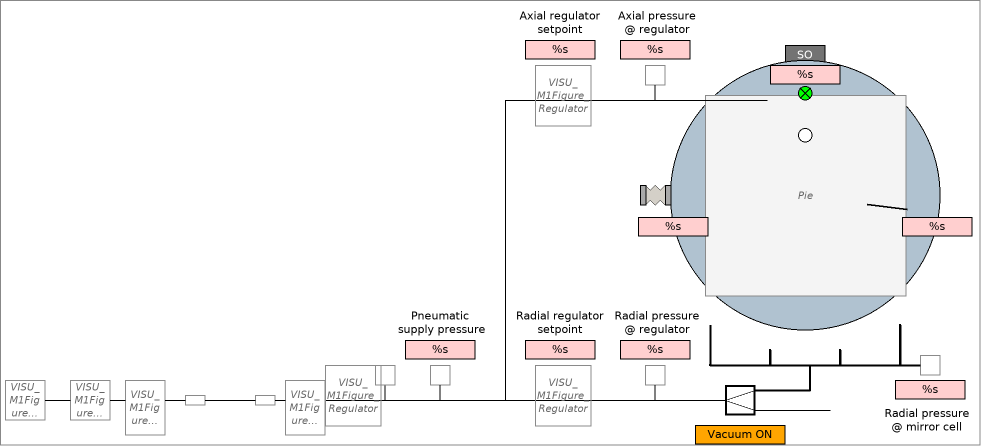
VISUALIZATION VISU_M1Figure  // 981x446
VAR_IN_OUT
	ref : M1;
    widget : M1Widget;
END_VAR
    Rectangle (785,45 40x33), "NW"
        p2858320360: widget.figure.axialNorthWestAngle
    Rectangle (785,45 40x30), "NE"
        p2858320360: widget.figure.axialNorthEastAngle
    Rectangle (785,45 40x33), "SO"
        p2858320360: widget.figure.axialSouthAngle
    Ellipse (670,60 270x270)
    Ellipse (770,160 70x70)
    Frame (920,355 20x20)
        shows VISU_M1Figure_Gauge()
    Rectangle (895,380 70x19), "%s", text variable: widget.figure.radialMirrorPressureString, colour variable: widget.radialSupport.mirrorPressure.actualStatusWidget.color.bg
        p55702900: widget.radialSupport.mirrorPressure.actualStatusWidget.color.fg
    Label (875,400 104x40), "Radial pressure @ mirror cell"
    Rectangle (725,385 30x30)
    Polyline (710,325) (710,365) (770,365) (770,350) (770,365) (840,365) (840,350) (840,365) (900,365) (900,325) (900,365) (920,365)
    Polyline (755,390) (810,390) (810,365)
    Rectangle (695,425 90x19), "Vacuum OFF", invisible if: ref.parts.radialSupport.parts.vacuumRelay.digitalOutput
    Line (755,410) (810,410)
    Line (810,410) (830,410)
    Line (725,400) (755,390), invisible if: ref.parts.radialSupport.parts.vacuumRelay.digitalOutput
    Line (725,400) (755,410), invisible if: NOT ref.parts.radialSupport.parts.vacuumRelay.digitalOutput
    Line (325,400) (725,400)
    Rectangle (665,185 6x20)
        p2858320360: widget.figure.radPad0Angle
    Polygon (650,200) (645,205) (645,185) (650,190) (655,185) (660,190) (665,185) (665,205) (660,200) (655,205)
        p2858320360: widget.figure.radPad0Angle
    Rectangle (640,185 6x20)
        p2858320360: widget.figure.radPad0Angle
    Rectangle (665,185 6x20)
        p2858320360: widget.figure.radPad1Angle
    Polygon (650,200) (645,205) (645,185) (650,190) (655,185) (660,190) (665,185) (665,205) (660,200) (655,205)
        p2858320360: widget.figure.radPad1Angle
    Rectangle (640,185 6x20)
        p2858320360: widget.figure.radPad1Angle
    Rectangle (665,185 6x20)
        p2858320360: widget.figure.radPad2Angle
    Polygon (650,200) (645,205) (645,185) (650,190) (655,185) (660,190) (665,185) (665,205) (660,200) (655,205)
        p2858320360: widget.figure.radPad2Angle
    Rectangle (640,185 6x20)
        p2858320360: widget.figure.radPad2Angle
    Rectangle (665,185 6x20)
        p2858320360: widget.figure.radPad3Angle
    Polygon (650,200) (645,205) (645,185) (650,190) (655,185) (660,190) (665,185) (665,205) (660,200) (655,205)
        p2858320360: widget.figure.radPad3Angle
    Rectangle (640,185 6x20)
        p2858320360: widget.figure.radPad3Angle
    Ellipse (744,135 123x123)
    Pie (705,95 201x201)
    Polyline (867,204) (907,209)
        p2858320360: widget.figure.axialSouthAngle
    Pie (705,95 201x201)
    Polyline (867,204) (907,209)
        p2858320360: widget.figure.axialNorthEastAngle
    Pie (705,95 201x201)
    Polyline (867,204) (907,209)
        p2858320360: widget.figure.axialNorthWestAngle
    Ellipse (798,128 14x14)
        p2858320360: widget.figure.axPadInner0Angle
    Ellipse (798,128 14x14)
        p2858320360: widget.figure.axPadInner1Angle
    Ellipse (798,128 14x14)
        p2858320360: widget.figure.axPadInner2Angle
    Ellipse (798,128 14x14)
        p2858320360: widget.figure.axPadInner3Angle
    Ellipse (798,128 14x14)
        p2858320360: widget.figure.axPadInner4Angle
    Ellipse (798,128 14x14)
        p2858320360: widget.figure.axPadInner5Angle
    Rectangle (770,65 70x19), "%s", text variable: widget.figure.axialForceStringSO, colour variable: widget.axialSupport.mirrorSouthForce.actualStatusWidget.color.bg
        p55702900: widget.axialSupport.mirrorSouthForce.actualStatusWidget.color.fg
    Rectangle (638,217 70x19), "%s", text variable: widget.figure.axialForceStringNW, colour variable: widget.axialSupport.mirrorNorthWestForce.actualStatusWidget.color.bg
        p55702900: widget.axialSupport.mirrorNorthWestForce.actualStatusWidget.color.fg
    Rectangle (902,217 70x19), "%s", text variable: widget.figure.axialForceStringNE, colour variable: widget.axialSupport.mirrorNorthEastForce.actualStatusWidget.color.bg
    Ellipse (798,86 14x14)
        p2858320360: widget.figure.axPad0Angle
    Ellipse (798,86 14x14)
        p2858320360: widget.figure.axPad1Angle
    Ellipse (798,86 14x14)
        p2858320360: widget.figure.axPad2Angle
    Ellipse (798,86 14x14)
        p2858320360: widget.figure.axPad3Angle
    Ellipse (798,86 14x14)
        p2858320360: widget.figure.axPad4Angle
    Ellipse (798,86 14x14)
        p2858320360: widget.figure.axPad5Angle
    Ellipse (798,86 14x14)
        p2858320360: widget.figure.axPad6Angle
    Ellipse (798,86 14x14)
        p2858320360: widget.figure.axPad7Angle
    Ellipse (798,86 14x14)
        p2858320360: widget.figure.axPad8Angle
    Ellipse (798,86 14x14), colour variable: widget.axialSupport.mirrorSouthForce.actualStatusWidget.color.bg
        p2858320360: widget.figure.axialSouthAngle
        p55702900: widget.axialSupport.mirrorSouthForce.actualStatusWidget.color.bg
    Polyline (810,98) (800,88)
        p2858320360: widget.figure.axialSouthAngle
    Polyline (810,88) (800,98)
        p2858320360: widget.figure.axialSouthAngle
    Ellipse (798,86 14x14), colour variable: widget.axialSupport.mirrorNorthEastForce.actualStatusWidget.color.bg
        p2858320360: widget.figure.axialNorthEastAngle
    Polyline (810,98) (800,88)
        p2858320360: widget.figure.axialNorthEastAngle
    Polyline (810,88) (800,98)
        p2858320360: widget.figure.axialNorthEastAngle
    Ellipse (798,86 14x14), colour variable: widget.axialSupport.mirrorNorthWestForce.actualStatusWidget.color.bg
        p2858320360: widget.figure.axialNorthWestAngle
    Polyline (810,98) (800,88)
        p2858320360: widget.figure.axialNorthWestAngle
    Polyline (810,88) (800,98)
        p2858320360: widget.figure.axialNorthWestAngle
    Line (505,100) (767,100)
    Frame (645,65 20x20)
        shows VISU_M1Figure_Gauge()
    Line (655,100) (655,85)
    Rectangle (620,40 70x19), "%s", text variable: widget.figure.axialRegulatorPressureString, colour variable: widget.axialSupport.regulatorPressure.actualStatusWidget.color.bg
        p55702900: widget.axialSupport.regulatorPressure.actualStatusWidget.color.fg
    Label (605,5 104x35), "Axial pressure @ regulator"
    Frame (535,65 56x61)
        shows VISU_M1Figure_Regulator()
    Label (515,5 90x35), "Axial regulator setpoint"
    Rectangle (525,40 70x19), "%s", text variable: widget.figure.axialRegulatorSetpointString, colour variable: widget.axialSupport.actualStatus.color.bg
        p55702900: widget.axialSupport.actualStatus.color.fg
    Frame (645,365 20x20)
        shows VISU_M1Figure_Gauge()
    Line (655,400) (655,385)
    Rectangle (620,340 70x19), "%s", text variable: widget.figure.radialRegulatorPressureString, colour variable: widget.radialSupport.regulatorPressure.actualStatusWidget.color.bg
        p55702900: widget.radialSupport.regulatorPressure.actualStatusWidget.color.fg
    Label (605,305 104x35), "Radial pressure @ regulator"
    Frame (535,365 56x61)
        shows VISU_M1Figure_Regulator()
    Label (515,305 90x35), "Radial regulator setpoint"
    Rectangle (525,340 70x19), "%s", text variable: widget.figure.radialRegulatorSetpointString, colour variable: widget.radialSupport.actualStatus.color.bg
        p55702900: widget.radialSupport.actualStatus.color.fg
    Line (505,100) (505,400)
    Frame (430,365 20x20)
        shows VISU_M1Figure_Gauge()
    Line (440,400) (440,385)
    Label (390,305 104x35), "Pneumatic supply pressure"
    Rectangle (405,340 70x19), "%s", text variable: widget.figure.supplyPressureString, colour variable: widget.pneumaticSupplyPressure.actualStatusWidget.color.bg
        p55702900: widget.pneumaticSupplyPressure.actualStatusWidget.color.fg
    Line (385,400) (385,385)
    Frame (375,365 20x20)
        shows VISU_M1Figure_Gauge()
    Frame (325,365 56x61)
        shows VISU_M1Figure_Regulator()
    Frame (255,395 20x10)
        shows VISU_M1Figure_Valve()
    Frame (285,380 40x55)
        shows VISU_M1Figure_FilterWithDrain()
    Line (215,400) (245,400)
    Frame (5,380 40x40)
        shows VISU_M1Figure_Supply()
    Frame (185,395 20x10)
        shows VISU_M1Figure_Valve()
    Frame (125,380 40x55)
        shows VISU_M1Figure_FilterWithDrain()
    Frame (70,380 40x40)
        shows VISU_M1Figure_Dryer()
    Rectangle (695,425 90x19), "Vacuum ON", invisible if: NOT ref.parts.radialSupport.parts.vacuumRelay.digitalOutput
    Line (275,400) (285,400)
    Line (245,400) (255,400)
    Line (205,400) (215,400)
    Line (165,400) (185,400)
    Line (110,400) (125,400)
    Line (45,400) (70,400)
END_VISUALIZATION

(* stored: Version 1.1.0.1, ProductVersion 3.1.4019.2
   Visu VISU_M1Figure: Id {eb73ebbd-d28e-47f1-8421-a160051d7996} *)
